RoboDK station: Robot_file.rdk

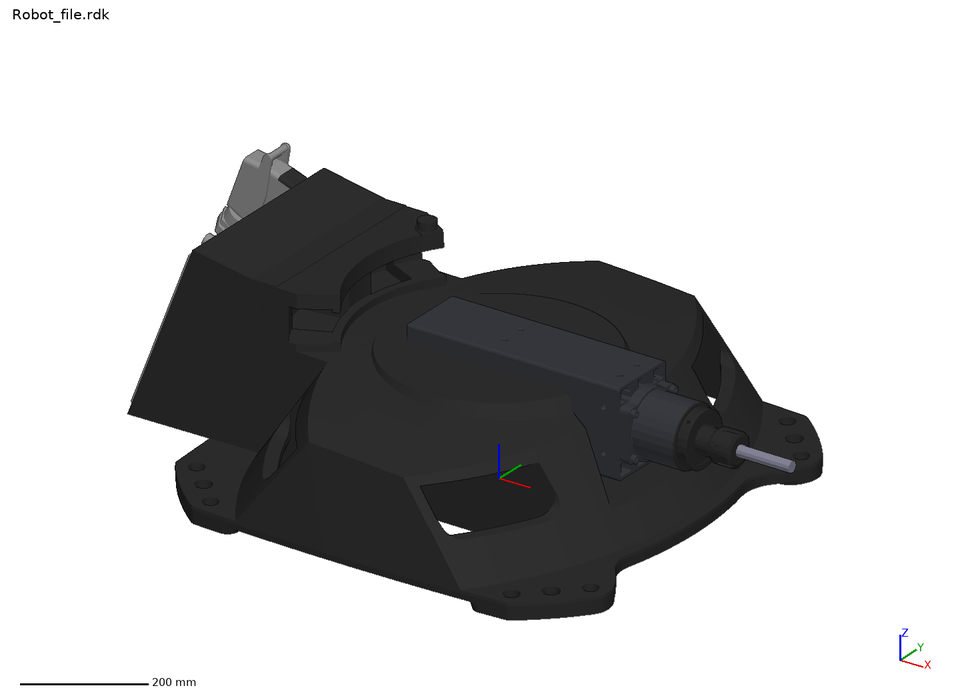
[picture v0: the station drawn from its stored meshes, robots at their saved joint values, targets as dots, program paths as lines]
Station Robot_file (saved by RoboDK 5.2.3). Poses are relative to the parent item; angles as X-Y-Z fixed-axis rotations.
  - frame KUKA KR 210 R2700 extra Base at (0, 0, 0) mm
    - frame Frame_2 at (1500, 1000, 500) mm
    - robot KUKA KR 210 R2700 extra: 6 axes, payload 210 kg, reach 2696 mm, repeatability 0.06 mm, weight 1068 kg
        joint limits [-185, -140, -120, -350, -125, -350] to [185, -5, 155, 350, 125, 350]; home [0, -90, 90, 0, 0, 0]; saved at [-34.544, -65.789, 91.833, 122.53, 42.264, -130.756]
      - tool Spindle, TCP at (557.2, 0, 176) mm, rotated rx 0 ry 90 rz 0 deg, size 692.9 x 170 x 256 mm
  - Python program FinalRobotPlan (listed below)

--- Python program FinalRobotPlan ---
'''
P_START = [1755, -500, 2155]
P_END   = [1755,  600, 2155]
NUM_POINTS  = 10


def MakePoints(xStart, xEnd, numPoints):
    if len(xStart) != 3 or len(xEnd) != 3:
        raise Exception("Start and end point must be 3-dimensional vectors")
    if numPoints < 2:
        raise Exception("At least two points are required")


    pt_list = []
    x = xStart[0]
    y = xStart[1]
    z = xStart[2]


    x_steps = (xEnd[0] - xStart[0])/(numPoints-1)
    y_steps = (xEnd[1] - xStart[1])/(numPoints-1)
    z_steps = (xEnd[2] - xStart[2])/(numPoints-1)


    for i in range(numPoints):
        point_i = [x,y,z]

        pt_list.append(point_i)
        x = x + x_steps
        y = y + y_steps
        z = z + z_steps
    return pt_list




POINTS = MakePoints(P_START, P_END, NUM_POINTS)
'''
from robolink import *
from robodk import *

data = open('wingbox_robodk_coordinates generator txt formatted.txt')
POINTS = []




# read table and get rid of fat
for line in data:
    row = line.split('\t')
    rowclean = []
    for item in row:
        item.strip('\t')
        if item == '':
            pass
        else:
            rowclean.append(item)
    del rowclean[3]
    res = [float(i) for i in rowclean]
    POINTS.append(res)





print(POINTS)
RDK = Robolink()


RDK.Render(False)


list_items = RDK.ItemList()
for item in list_items:
    if item.Name().startswith('Auto'):
        item.Delete()


robot = RDK.ItemUserPick('Select a robot', ITEM_TYPE_ROBOT)


RDK.Render(True)


if not robot.Valid():
    quit()

'''
RDK.AddFrame("Frame")
RDK.setPose(transl(100,200,300) * rotz(pi/2))
'''
reference = robot.Parent()


robot.setPoseFrame(reference)


pose_ref = robot.Pose()
print(Pose_2_TxyzRxyz(pose_ref))





for i in range(len(POINTS)):

    pose_i = pose_ref
    pose_i.setPos(POINTS[i])


    robot.MoveJ(pose_i)


quit()
